
TYPE "AlarmConfig_001"
STRUCT
        ENABLED : BOOL;
        PRIORITY : INT;
        DELAY_TIME : TIME;
        MESSAGE : STRING;
        ACKNOWLEDGEMENT_REQUIRED : BOOL;
        ALARM_CLASS : INT;
        ALARM_GROUP : INT;
END_STRUCT;
END_TYPE